# EPICS autosave request: acsMotionApp/Db/SPiiPlusMaxParams_settings.req
$(P)$(M):maxVelocity.VAL
$(P)$(M):maxVelocity.PREC
$(P)$(M):maxAcceleration.VAL
$(P)$(M):maxAcceleration.PREC
